// Mitsubishi GX Works2 project: PT100_G2   PLC: Q03UDE

PROGRAM MAIN
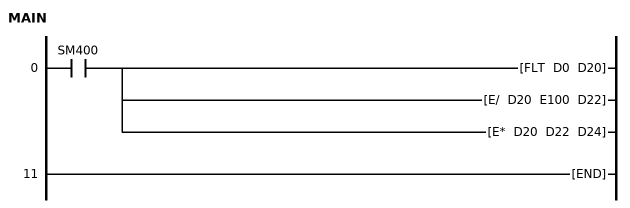
0     LD      SM400
      FLT     D0 D20
      E/      D20 E100 D22
      E*      D20 D22 D24
11    END
END_PROGRAM
